FUNCTION_BLOCK EDCA
  (* Standard: 61499-2 *)
  (* Version 0.1, 2015-00-24, Jin, Jin-PC *)
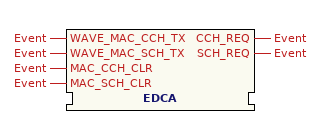
  EVENT_INPUT
    WAVE_MAC_CCH_TX;
    WAVE_MAC_SCH_TX;
    MAC_CCH_CLR;
    MAC_SCH_CLR;
  END_EVENT
  EVENT_OUTPUT
    CCH_REQ;
    SCH_REQ;
  END_EVENT
END_FUNCTION_BLOCK
(* other elements stored in the file *)
(* ECC Name=EDCA *)
(* ECState Name=EDCA *)
(* ECC Name=bufferCCH *)
(* ECState Name=CCHempty *)
(* ECState Name=CCHfull *)
(* ECAction Output=CCH_REQ *)
(* ECTransition Source=CCHempty Destination=CCHfull Condition=WAVE_MAC_CCH_TX *)
(* ECTransition Source=CCHfull Destination=CCHempty Condition=MAC_CCH_CLR *)
(* ECTransition Source=CCHfull Destination=CCHfull Condition=true *)
(* ECC Name=bufferSCH *)
(* ECState Name=SCHempty *)
(* ECState Name=SCHfull *)
(* ECAction Output=SCH_REQ *)
(* ECTransition Source=SCHempty Destination=SCHfull Condition=WAVE_MAC_SCH_TX *)
(* ECTransition Source=SCHfull Destination=SCHempty Condition=MAC_SCH_CLR *)
(* ECTransition Source=SCHfull Destination=SCHfull Condition=true *)
